// TwinCAT 3 PLC project PLC2
// ProgramVersion: 3.1.4024.0
// libraries:
//   Tc2_Standard, * (Beckhoff Automation GmbH)
//   Tc2_System, * (Beckhoff Automation GmbH)
//   Tc3_Module, * (Beckhoff Automation GmbH)
//   VisuSymbols,3.5.10.0,System
// project tree:
//   / GlobalTextList.TcGTLO, PlcTask.TcTTO, Task_PRG1.TcTTO, Task_PRG2.TcTTO, Visualization Manager.TcVMO (not stored)
//   GVLs/ GVL.TcGVL
//   POUs/ FC1_Bereken_Snelheid.TcPOU, MAIN.TcPOU, PRG1_Conveyer_Operation.TcPOU, PRG2_Object_Detectie.TcPOU
//   VISUs/ Overview.TcVIS
// real-time tasks:
//   TASK PlcTask: cycle T#10ms, priority 20, ADS port 350
//   TASK Task_PRG1: cycle T#100000us, priority 1, ADS port 351
//   TASK Task_PRG2: cycle T#1000ms, priority 2, ADS port 352

CONFIGURATION PLC2
    RESOURCE PLC ON TwinCAT3
        TASK PlcTask(INTERVAL := T#10ms, PRIORITY := 20);
        TASK Task_PRG1(INTERVAL := T#100000us, PRIORITY := 1);
        TASK Task_PRG2(INTERVAL := T#1000ms, PRIORITY := 2);
        PROGRAM MAIN WITH PlcTask : MAIN;
        PROGRAM PRG1_Conveyer_Operation WITH Task_PRG1 : PRG1_Conveyer_Operation;
        PROGRAM PRG2_Object_Detectie WITH Task_PRG2 : PRG2_Object_Detectie;
    END_RESOURCE
END_CONFIGURATION

// ---- GVLs/GVL.TcGVL
{attribute 'qualified_only'}
VAR_GLOBAL

// Hele rits aan variabelen

// -----------------------------------------Ingangen	
// Digitale Ingangen
	KN_001 			AT%IX0.0 : BOOL := 0;  // systeem opstartknop
	KN_002 			AT%MX0.1 : BOOL := 0;  // Acknowledge All Alarms -- 	(MX om de knop weer laag te schrijven, kan niet naar IX schrijven ¯\_(ツ)_/¯  )
	In2Res 			AT%IX0.2 : BOOL := 0;  // Reserve
	In3Res 			AT%IX0.3 : BOOL := 0;  // Reserve 
	In4Res 			AT%IX0.4 : BOOL := 0;  // Reserve 
	LS_001 			AT%MX0.5 : BOOL := 0;  // objectdetectie sensor weegcel (MX om d.m.v. timer laag te schrijven, kan niet naar IX schrijven ¯\_(ツ)_/¯  )
	LS_002 			AT%IX0.6 : BOOL := 0;  // objectdetectie sensor eind van transportbaan 
	In7Res 			AT%IX0.7 : BOOL := 0;  // Reserve 
	In8Res 			AT%IX1.0 : BOOL := 0;  // Reserve 
	In9Res 			AT%IX1.1 : BOOL := 0;  // Reserve
	
// Analoge ingangen 
	weegcelWaarde 	AT%IW10 : DINT := 1;  // ingelezen gewicht van de lading 
	In11Res 		AT%IW12 : DINT := 0;  // Reserve
	In12Res 		AT%IW14 : DINT := 0;  // Reserve
	In13Res 		AT%IW16 : DINT := 0;  // Reserve 
	In14Res 		AT%IW18 : DINT := 0;  // Reserve 
	In15Res 		AT%IW20 : DINT := 0;  // Reserve 
	In16Res 		AT%IW22 : DINT := 0;  // Reserve
	In17Res 		AT%IW24 : DINT := 0;  // Reserve
	In18Res 		AT%IW26 : DINT := 0;  // Reserve
	In19Res 		AT%IW28 : DINT := 0;  // Reserve
	
// -----------------------------------------Uitgangen
// Digitale Uitgangen
	transportActief 	AT%QX0.0 : BOOL := 0;  // transportbaan aangezet signaal
	alarmActief 		AT%QX0.1 : BOOL := 0;  // alarm melding
	Uit2Res 			AT%QX0.2 : BOOL := 0;  // Reserve
	Uit3Res 			AT%QX0.3 : BOOL := 0;  // Reserve
	Uit4Res 			AT%QX0.4 : BOOL := 0;  // Reserve
	Uit5Res 			AT%QX0.5 : BOOL := 0;  // Reserve
	Uit6Res 			AT%QX0.6 : BOOL := 0;  // Reserve
	Uit7Res 			AT%QX0.7 : BOOL := 0;  // Reserve
	Uit8Res 			AT%QX1.0 : BOOL := 0;  // Reserve
	Uit9Res 			AT%QX1.1 : BOOL := 0;  // Reserve

// Analoge Uitgangen 
	geschrevenSnelheid 		AT%QW10 : DINT := 0;  // snelheid uitgeschreven naar motor
	Uit11Res 				AT%QW12 : DINT := 0;  // Reserve
	Uit12Res				AT%QW14 : DINT := 0;  // Reserve
	Uit13Res 				AT%QW16 : DINT := 0;  // Reserve
	Uit14Res 				AT%QW18 : DINT := 0;  // Reserve
	Uit15Res 				AT%QW20 : DINT := 0;  // Reserve
	Uit16Res 				AT%QW22 : DINT := 0;  // Reserve
	Uit17Res 				AT%QW24 : DINT := 0;  // Reserve
	Uit18Res 				AT%QW26 : DINT := 0;  // Reserve 
	Uit19Res 				AT%QW28 : DINT := 0;  // Reserve


// Globale Variabelen
// Bool Statussen
	systeemStatus 			AT%MX0.0 : BOOL := 0; // 0 = uit, 1 = actief
	objectDetected			AT%MX0.1 : BOOL := 0;
	ALM001					AT%MX0.2 : BOOL := 0; // missend object - alarm
	
// INT&DINT&REAL opslag
	PRG1_Status				AT%MW10 : INT := 0; 	// 0 = idle, 1 = running, 2 = fault	
	ladingGewicht 			AT%MW12 : DINT := 0; 	// opslag gelezen gewicht
	berekendeSnelheid		AT%MW14 : DINT;
	transportBaanVoortgang 	AT%MW16 : DINT;
	transportBaanEinde		AT%MW18 : UINT := 800;
//	cyclusTijd				AT%MW20 : TIME := T#10MS;
	
	//variabelen voor snelheidberekening

	
	
END_VAR

// ---- POUs/MAIN.TcPOU
PROGRAM MAIN
VAR
	
END_VAR

(*
	BOUW  Alarm als berekende snelheid == 0;




*)



//PRG1_Conveyer_Operation();
//PRG2_Object_Detectie();

END_PROGRAM

// ---- POUs/PRG1_Conveyer_Operation.TcPOU
PROGRAM PRG1_Conveyer_Operation
VAR_INPUT
	
END_VAR
VAR
	weegTijd 			: INT 			:= 0;
	weegEind 			: INT 			:= 50;
	runningTijd  		: INT 			:= 0;
	detectieLaagTijd  	: INT 			:= 40;
	alarmTijd			: INT			:= 0;
	Modus				: STRING(INT#8) := 'OFF';
	voortangDeling		: INT			:= 100;
	checkpunt			: INT 			:= 0;
END_VAR


// Read startknop
IF NOT GVL.KN_001 AND NOT GVL.alarmActief THEN
	GVL.PRG1_Status := 0;
	GVL.transportActief := FALSE;
END_IF

//als alarm dan naar FAULT
IF NOT GVL.KN_001 AND GVL.alarmActief THEN
	GVL.PRG1_Status := 3;
END_IF

//case functie, voor conveyerstatussen
CASE GVL.PRG1_Status OF
	0:	// OFF, wacht op startknop
		Modus := 'OFF';
		
		IF GVL.KN_001 THEN
			GVL.PRG1_Status := 1;
		END_IF
	1: // idle, wacht op object	
		Modus := 'IDLE';
		
		//reset berekening voor volgende weging
		GVL.berekendeSnelheid := 0;
		
		// als no object detected berekent FC1 de maximale tijd tot alarm
		IF GVL.objectDetected = TRUE THEN
			
			weegTijd := weegTijd + 2;
			GVL.ladingGewicht := GVL.weegcelWaarde;								
			GVL.berekendeSnelheid := FC1_Bereken_Snelheid(GVL.ladingGewicht);//GVL.MinGewicht, GVL.MaxGewicht,GVL.MinSpeed,GVL.MaxSpeed
			IF weegTijd >= weegEind THEN
				GVL.PRG1_Status := 2;
				//reset weegtijd
				weegTijd := 0;
			END_IF
			
		END_IF
		
	2: //running
		Modus := 'RUNNING';
		
		GVL.transportActief := TRUE;
		GVL.geschrevenSnelheid := GVL.berekendeSnelheid;
			
		// Runtijd tellen
		runningTijd := runningTijd + 10;
		
		IF runningTijd > 4 THEN // reset sensor
			GVL.LS_001 := FALSE;
		END_IF
		
		// Tijd conversie naar transportbaan voortgang.
		GVL.transportBaanVoortgang := GVL.geschrevenSnelheid * (runningTijd/voortangDeling);
		
		// Vergelijk voortgang met einde transportbaan, vervolgens reset waarden en status naar IDLE
		IF GVL.transportBaanVoortgang >= GVL.transportBaanEinde THEN
			GVL.transportActief := FALSE;
			GVL.transportBaanVoortgang := 0;
			GVL.geschrevenSnelheid := 0; 
			runningTijd := 0;
			GVL.PRG1_Status := 1;
		END_IF
		
	3: // Fault
		Modus := 'FAULT';
		IF GVL.KN_002 THEN
			GVL.alarmActief := FALSE;
			GVL.PRG1_Status := 1;
		END_IF
END_CASE

END_PROGRAM

// ---- POUs/FC1_Bereken_Snelheid.TcPOU
FUNCTION FC1_Bereken_Snelheid : DINT

VAR_INPUT
    Laadgewicht : DINT;    // Invoer van de weegcel
END_VAR

VAR
    // Definieer de minimale en maximale gewichten en snelheden
    MinGewicht  : REAL := 1.0;    // Minimum gewicht
    MaxGewicht  : REAL := 100.0;  // Maximum gewicht
    MinSpeed    : REAL := 50.0;    // Minimum snelheid
    MaxSpeed    : REAL := 200.0;  // Maximum snelheid

    BerekendeSnelheid : REAL;     // De berekende snelheid in REAL
    LaadgewichtReal   : REAL;     // Laadgewicht geconverteerd naar REAL
END_VAR



// Converteer Laadgewicht naar REAL voor de berekening
LaadgewichtReal := DINT_TO_REAL(Laadgewicht);

// Controleer of Laadgewicht binnen het verwachte bereik valt
IF LaadgewichtReal < MinGewicht THEN
    LaadgewichtReal := MinGewicht;  // Zorg dat het gewicht niet lager is dan MinGewicht
ELSIF LaadgewichtReal > MaxGewicht THEN
    LaadgewichtReal := MaxGewicht;  // Zorg dat het gewicht niet hoger is dan MaxGewicht
END_IF

// Bereken de snelheid op basis van het gewicht
BerekendeSnelheid := MaxSpeed - ((LaadgewichtReal - MinGewicht) / (MaxGewicht - MinGewicht) * (MaxSpeed - MinSpeed));

// Rond de berekende snelheid af naar een DINT waarde en retourneer deze
FC1_Bereken_Snelheid := REAL_TO_DINT(BerekendeSnelheid);

END_FUNCTION

// ---- POUs/PRG2_Object_Detectie.TcPOU
PROGRAM PRG2_Object_Detectie
VAR
    ObjectAanwezig : BOOL;    			// Invoer van de sensor, TRUE als object gedetecteerd
    AlarmStatus    : BOOL;    			// Uitvoer, TRUE als er geen object is gedetecteerd
    MaxWachttijd   : INT := 30;    	// Maximale tijd om te wachten op een object
    Wachttijd      : INT := 0;    			// Huidig wachttijd zonder objectdetectie
END_VAR



// lezen ingangen
ObjectAanwezig := GVL.LS_001; 


//reset wachttijd met alarm acknowledge
IF GVL.KN_002 THEN
	Wachttijd := 0;
	AlarmStatus := FALSE;
END_IF

IF GVL.PRG1_Status = 1 THEN
	// Controleer of een object aanwezig is op de transportband
	IF ObjectAanwezig = TRUE THEN
		// Object gedetecteerd, reset de wachttijd en schakel het alarm uit
		Wachttijd := 0;
		AlarmStatus := FALSE;
	ELSE//wacht op detectie, tot maximale tijd verstreken en alarm geactiveerd
		// Geen object gedetecteerd, verhoog de wachttijd
			
		Wachttijd := Wachttijd + 1;  // Verhoog de gewachtte tijd per cyclus 
	
		// Activeer het alarm als de wachttijd de maximale tijd overschrijdt
		IF Wachttijd >= MaxWachttijd THEN
			AlarmStatus := TRUE;
			GVL.PRG1_Status := 3;
		END_IF
	END_IF
END_IF


//stuur statussen naar GVL.
GVL.objectDetected  :=  ObjectAanwezig;	
GVL.ALM001 			:= 	AlarmStatus; 	// schrijven in geheugen voor OPC/SCADA of weet ik het wat nog meer.
GVL.alarmActief 	:= 	AlarmStatus;	// sturen naar digitale uitgang

END_PROGRAM

// ---- GlobalTextList.TcGTLO
TEXTLIST GlobalTextList
  524 = '%s'
  391 = 'Acknowledge'
  561 = 'Alarm001'
  960 = 'Berekend: %i'
  427 = 'Current State : %i'
  497 = 'Current State : %s'
  584 = 'Detectie & weging'
  904 = 'Gestuurd: %i'
  996 = 'Startknop'
  150 = 'TransportActief'
  118 = 'Weegschaal'
  675 = 'WEEGSCHAAL'
END_TEXTLIST

// ---- VISUs/Overview.TcVIS
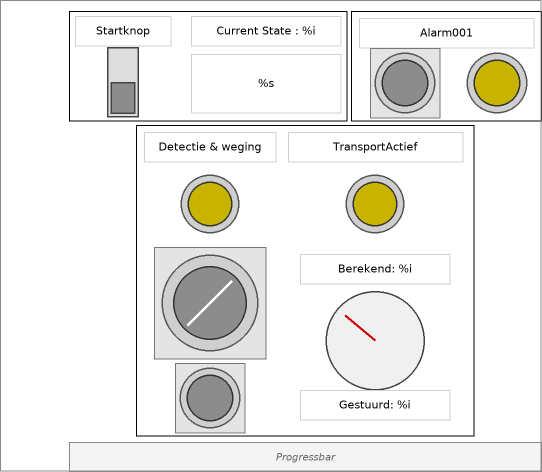
VISUALIZATION Overview  // 542x472
    Progressbar (69,442 473x30), variable: GVL.transportBaanVoortgang
    Rectangle (136,125 338x311)
    Potentiometer360 (154,243 112x120), variable: GVL.weegcelWaarde, style: Potentiometer-Potentiometer360-Gray, scale format: %.1f, scale 0..100
        p2431819421: Outside
    PushSwitchLed (175,363 70x70), variable: GVL.LS_001, behaviour: TOGGLE, style: Switch-PushSwitchLed-Gray
    Lamp1 (176,169 68x70), variable: GVL.objectDetected, style: Lamp-Lamp1-Yellow
    Textfield (144,132 132x30), "Detectie & weging"
    Group (277,254 196x166)
        Textfield (23,0 150x30), "Berekend: %i", text variable: GVL.berekendeSnelheid
        Group (0,37 196x129)
            Meter180 (0,0 196x99), value: GVL.snelheidSetpoint, style: Meter-Meter180-Gray, scale format: %.1f, scale 0..200
            Textfield (23,99 150x30), "Gestuurd: %i", text variable: GVL.snelheidSetpoint
    Lamp1 (341,169 68x70), variable: GVL.transportActief, style: Lamp-Lamp1-Yellow
    Textfield (288,132 175x30), "TransportActief"
    Rectangle (351,11 191x110)
    Textfield (359,18 175x30), "Alarm001"
    Lamp1 (462,48 70x70), variable: GVL.alarmActief, style: Lamp-Lamp1-Yellow
    PushSwitch (370,48 70x70), variable: GVL.KN_002, behaviour: TOGGLE, style: Switch-PushSwitch-Gray
    Rectangle (69,11 278x110)
    Textfield (75,16 96x30), "Startknop"
    DipSwitch (88,47 70x70), variable: GVL.KN_001, behaviour: TOGGLE, style: Switch-DipSwitch-Gray
    Textfield (191,16 150x30), "Current State : %i", text variable: GVL.PRG1_Status
    Textfield (191,54 150x59), "%s", text variable: PRG1_Conveyer_Operation.Modus
END_VISUALIZATION
